Fanuc KAREL source: IO0108.KL

-- PROVISIONAL review KL for V1013-1; original PC SHA256 66a4d84fb191b89d5f755ff3f98c1748127e9e55595e0f94883746ac4309f830
-- Incomplete behavior may be omitted. Consult companion uncertainty JSON. Do not deploy.
PROGRAM IO0108
%NOLOCKGROUP
-- UNRESOLVED_LOCAL_POOL 5 cells at code offset 13; source declarations unknown
-- DIRECT_LOCAL_WORD_ACCESS alone does not prove INTEGER, REAL, or BOOLEAN
BEGIN
  -- UNRESOLVED_PC offsets 0-18; opcodes 2B,2C,7B
  -- UNRESOLVED_PC offsets 23-30; opcodes 9D,23
  -- UNRESOLVED_PC offsets 35-49; opcodes 2E,22,9D,33,35
  -- UNRESOLVED_PC offsets 54-61; opcodes 9D,23
  -- UNRESOLVED_PC offsets 66-77; opcodes 2E,23
  -- UNRESOLVED_PC offsets 82-91; opcodes 21,9D,1A
  -- UNRESOLVED_PC offsets 96-100; opcodes 7F
  -- UNRESOLVED_PC offsets 105-109; opcodes 27,AA
  -- UNRESOLVED_PC offsets 114-118; opcodes 7F
END IO0108
